{attribute 'qualified_only'}
TYPE EDataType :
(
	none := 0,
	dont_care := 1,
	binary := 2,
	numeric := 3,
	string_t := 4
) USINT;
END_TYPE

(* stored: Version 1.1.0.1
   DUT EDataType: Id {c7181a47-a5ea-4063-9a72-ca9ae11cbe72} *)
